INTERFACE ITF_BaseControlElement_HMI_Connector EXTENDS 
		ITF_BaseControlElement_HMI_Connector_View, ITF_BaseControlElement_HMI_Connector_Command

END_INTERFACE

(* stored: Version 1.1.0.1
   Itf ITF_BaseControlElement_HMI_Connector: Id {bae10e73-0438-0fbc-0a7a-d25c1aa17aaf} *)
